// TIA Portal V18 export
FUNCTION_BLOCK "Simulation"   // FB1, FBD
TITLE = Simulation
{ S7_Optimized_Access := 'TRUE' }
AUTHOR : dda
VERSION : 0.1
// Simulate machine behaviour
// stored: AutoNumber true, IsIECCheckEnabled true, IsRetainMemResEnabled false, MemoryReserve 100, SetENOAutomatically true, UDAEnableTagReadback false
   VAR_INPUT
      moveUp { ExternalAccessible := 'False'; ExternalVisible := 'False'; ExternalWritable := 'False'} : Bool;
      moveDown { ExternalAccessible := 'False'; ExternalVisible := 'False'; ExternalWritable := 'False'} : Bool;
      MoveLeft { ExternalAccessible := 'False'; ExternalVisible := 'False'; ExternalWritable := 'False'} : Bool;
      moveRight { ExternalAccessible := 'False'; ExternalVisible := 'False'; ExternalWritable := 'False'} : Bool;
      runConveyor { ExternalAccessible := 'False'; ExternalVisible := 'False'; ExternalWritable := 'False'} : Bool;
      engineBroken { ExternalAccessible := 'False'; ExternalVisible := 'False'; ExternalWritable := 'False'} : Bool;
      robotGoToStation { ExternalAccessible := 'False'; ExternalVisible := 'False'; ExternalWritable := 'False'} : Bool;
      robotGoToMagazine { ExternalAccessible := 'False'; ExternalVisible := 'False'; ExternalWritable := 'False'} : Bool;
   END_VAR
   VAR_OUTPUT
      xPosition { ExternalAccessible := 'False'; ExternalVisible := 'False'; ExternalWritable := 'False'} : Int;
      yPosition { ExternalAccessible := 'False'; ExternalVisible := 'False'; ExternalWritable := 'False'} : Int;
      lightBeam1 { ExternalAccessible := 'False'; ExternalVisible := 'False'; ExternalWritable := 'False'} : Bool;
      lightBeam2 { ExternalAccessible := 'False'; ExternalVisible := 'False'; ExternalWritable := 'False'} : Bool;
      lightBeam3 { ExternalAccessible := 'False'; ExternalVisible := 'False'; ExternalWritable := 'False'} : Bool;
      robotPosHMI { ExternalAccessible := 'False'; ExternalVisible := 'False'; ExternalWritable := 'False'} : Int;
      robotHasChip { ExternalAccessible := 'False'; ExternalVisible := 'False'; ExternalWritable := 'False'} : Bool;
   END_VAR
   VAR
      instTimerSimulate { ExternalAccessible := 'False'; ExternalVisible := 'False'; ExternalWritable := 'False'; S7_SetPoint := 'True'} : TON_TIME;
      statSimulate { ExternalAccessible := 'False'; ExternalVisible := 'False'; ExternalWritable := 'False'} : Bool;
      StatPositionConveyor { ExternalAccessible := 'False'; ExternalVisible := 'False'; ExternalWritable := 'False'} : Int;
      statRobotHasChip { ExternalAccessible := 'False'; ExternalVisible := 'False'; ExternalWritable := 'False'} : Bool;
      statRobotPosHMI { ExternalAccessible := 'False'; ExternalVisible := 'False'; ExternalWritable := 'False'} : Int;
   END_VAR
   VAR_TEMP
      tempLB1 : Bool;
      tempLB2 : Bool;
      tempLB3 : Bool;
   END_VAR
   VAR CONSTANT
      SIMULATION_TIME : Time := T#10ms;
   END_VAR
BEGIN

REGION Network 1 (SCL)
   // Титульные комменты для блока
   // 
   // 22.12.2023
END_REGION

REGION Network 2: trigger simulation step
   // set bit one cycle every 10 ms
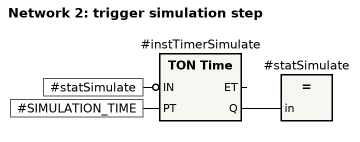
   #instTimerSimulate(IN := NOT #statSimulate, PT := #SIMULATION_TIME);   // TON
   #statSimulate := #instTimerSimulate.Q;
END_REGION

REGION Network 3 (SCL): Simulation step
   IF (#statSimulate = TRUE) AND (NOT #engineBroken) THEN
     // move robot
     IF #moveUp = TRUE THEN
       #yPosition += 1;
     END_IF;
     IF #moveDown = TRUE THEN
       #yPosition -= 1;
     END_IF;
     IF #MoveLeft = TRUE THEN
       #xPosition += 1;
     END_IF;
     IF #moveRight = TRUE THEN
       #xPosition -= 1;
     END_IF;
     // move conveyor
     IF (#StatPositionConveyor > 800) THEN
       #StatPositionConveyor := 0;
     ELSIF (#runConveyor = TRUE) THEN
       #StatPositionConveyor += 1;
     END_IF;
   END_IF;

   // for S7-300 / S7-400
   #tempLB1 := FALSE;
   #tempLB2 := FALSE;
   #tempLB3 := FALSE;

   // assign lightbeams
   CASE #StatPositionConveyor OF
     30..60:
       #tempLB1 := TRUE;
     500..530:
       #tempLB2 := TRUE;
     700..800:
       #tempLB3 := TRUE;

     ELSE   // Statement section ELSE
       ;
   END_CASE;

   #lightBeam1 := #tempLB1;
   #lightBeam2 := #tempLB2;
   #lightBeam3 := #tempLB3;

   // Calculate data for display of robot in HMI
   IF (#xPosition = 100)
   THEN
     #statRobotPosHMI := #yPosition;
   ELSE
     #statRobotPosHMI := 100;
   END_IF;
END_REGION
END_FUNCTION_BLOCK
